Yaskawa INFORM job: SCANNING_2.JBI

/JOB
//NAME SCANNING_2
//POS
///NPOS 15,0,15,1,0,1
///TOOL 0
///POSTYPE BASE
///RECTAN
///RCONF 0,0,0,0,0,0,0,0,0,0,0,0,0,0,0,0,0,0,0,0,0,0,0,0
C00000=1500.000,-700.000,-580.000,-100.0000,0.0000,-45.0000
C00001=1500.000,-700.000,-580.000,-100.0000,0.0000,-45.0000
C00002=1400.000,-800.000,0.000,-125.0000,0.0000,-45.0000
C00003=1400.000,-800.000,0.000,-125.0000,0.0000,-45.0000
C00004=1500.000,-700.000,-580.000,-100.0000,0.0000,-45.0000
C00005=1500.000,-700.000,-580.000,-100.0000,0.0000,-45.0000
C00006=1400.000,-800.000,0.000,-125.0000,0.0000,-45.0000
C00007=1400.000,-800.000,0.000,-125.0000,0.0000,-45.0000
C00008=1500.000,-700.000,-580.000,-100.0000,0.0000,-45.0000
C00009=1500.000,-700.000,-580.000,-100.0000,0.0000,-45.0000
C00010=1400.000,-800.000,0.000,-125.0000,0.0000,-45.0000
C00011=1400.000,-800.000,0.000,-125.0000,0.0000,-45.0000
C00012=1500.000,-700.000,-580.000,-100.0000,0.0000,-45.0000
C00013=1500.000,-700.000,-580.000,-100.0000,0.0000,-45.0000
C00014=1400.000,-800.000,0.000,-125.0000,0.0000,-45.0000
///POSTYPE PULSE
///PULSE
EC00000=0
EC00001=46080
EC00002=46080
EC00003=92160
EC00004=92160
EC00005=138240
EC00006=138240
EC00007=184620
EC00008=184620
EC00009=230400
EC00010=230400
EC00011=276480
EC00012=276480
EC00013=322560
EC00014=322560
///POSTYPE BASE
///RECTAN
P00002=1400.000,-800.000,0.000,-125.0000,0.0000,-45.0000
///POSTYPE PULSE
///PULSE
EX00000=0
//INST
///DATE 2023/01/30 09:59
///ATTR SC,RW,RJ
////FRAME BASE
///GROUP1 RB1,ST1
NOP
MOVJ P002 EX000 VJ=15.00
TIMER T=5.00
MOVL C00000 EC00000 V=350.0
TIMER T=1.00
MOVL C00001 EC00001 V=350.0
TIMER T=1.00
MOVL C00002 EC00002 V=350.0
TIMER T=1.00
MOVL C00003 EC00003 V=350.0
TIMER T=1.00
MOVL C00004 EC00004 V=350.0
TIMER T=1.00
MOVL C00005 EC00005 V=350.0
TIMER T=1.00
MOVL C00006 EC00006 V=350.0
TIMER T=1.00
MOVL C00007 EC00007 V=350.0
TIMER T=1.00
MOVL C00008 EC00008 V=350.0
TIMER T=1.00
MOVL C00009 EC00009 V=350.0
TIMER T=1.00
MOVL C00010 EC00010 V=350.0
TIMER T=1.00
MOVL C00011 EC00011 V=350.0
TIMER T=1.00
MOVL C00012 EC00012 V=350.0
TIMER T=1.00
MOVL C00013 EC00013 V=350.0
TIMER T=1.00
MOVL C00014 EC00014 V=350.0
MOVJ P002 VJ=15.00
END
